METHOD PUBLIC noAction : BOOL //Return value = TRUE if busy of home and motion 
VAR_INPUT
END_VAR
home.Execute	:= FALSE;


NoAction 		:= 	NOT home.Busy ;
END_METHOD

PROPERTY PUBLIC optEnableCmdAbortedAsError : BOOL
GET
optEnableCmdAbortedAsError := Options.7;
END_GET
SET
Options.7 := optEnableCmdAbortedAsError;
END_SET
END_PROPERTY

{attribute 'monitoring' := 'call'}
PROPERTY rAdmin : REFERENCE to AxAdmin
GET
rAdmin REF= Admin;
END_GET
END_PROPERTY

{attribute 'monitoring' := 'call'}
PROPERTY rAxisRef : REFERENCE TO AXIS_REF
GET
rAxisRef REF= THIS^;
END_GET
END_PROPERTY

{attribute 'monitoring' := 'call'}
PROPERTY PUBLIC rErrHdl : REFERENCE to ERROR_HDL
GET
rErrHdl REF= ErrHdl;
END_GET
SET
ErrHdl := rErrHdl;
END_SET
END_PROPERTY

METHOD reset : Bool
VAR_INPUT
END_VAR
NoAction();
reset 			:= ErrHdl.flag OR Admin.reset(FALSE);
Event.confirm();
END_METHOD

{attribute 'monitoring' := 'call'}
PROPERTY rHome : REFERENCE To AxHoming
GET
rHome REF= Home;
END_GET
END_PROPERTY

{attribute 'monitoring' := 'call'}
PROPERTY rPara : REFERENCE TO AxPara
GET
rPara REF= Para;
END_GET
END_PROPERTY

END_FUNCTION_BLOCK

// ---- POUs/Motion/TF5100-NCI/01_Main/NCI_REF.TcPOU
{attribute 'no_check'}
FUNCTION_BLOCK NCI_REF
VAR_INPUT
	PlcToNci										AT %Q*	: PLCTONC_NCICHANNEL_REF;	//link PLC to NC
END_VAR                             				
VAR_OUTPUT                          	
	NciToPlc										AT %I*	: NCTOPLC_NCICHANNEL_REF;	//link NC to PLC

(* Extrabits out of the struct *)
	ItpRunning												:	BOOL := FALSE;	//Interpreter is running
	ItpGroupActive											:	BOOL;			//Interpreter group is active -> Axes group build 			
	GrpCnfg													:	NCI_EXT3DGROUP;	//Group configuration
	                                    					
(* ChnState *******************)        					
	IsItpChn												:	BOOL := FALSE;	//TRUE when it is interpreter channel
	IsEStopRequested										:	BOOL := FALSE;	//TRUE when EStop is requested
	IsFeedFromBackupList									:	BOOL := FALSE;	//TRUE when parameter feed comes from backup list 
	IsMovingBackward										:	BOOL := FALSE;	//TRUE when moving forward
	
(* configurated parameters of the cyclic channel *)
	PathRestWay												:	LREAL;	//remaining arc length on the current path segment
	CurrentPathSetVelo										:	LREAL;	//current path set velocity
                                        					
	SAFStatus												:	UDINT;	//SAF state
	SAFEintraege											:	UDINT;	//current number of SAF entries/tasks
	SVBStatus												:	UDINT;	//SVB state
	SVBEintraege											:	UDINT;	//current number of SVB entries/tasks
	MemLastBlockNo											:	UDINT;	//contains last block number
END_VAR
VAR
	(* NciToPlc channel extend *)
	SetCyclicLrealOffsets									:	ItpSetCyclicLRealOffsets;
	SetCyclicLrealOffsetsDone								:	BOOL;
	SetCyclicUdintOffsets									:	ItpSetCyclicUdintOffsets;
	SetCyclicUdintOffsetsDone								:	BOOL;
	
END_VAR

;

METHOD readStatus : BOOL 
VAR_INPUT
END_VAR
(* NCI Status lesen															*)
(****************************************************************************)

(****************************************************************************)
(* 4 LReal variables to configurate the interface cyclely					*)
(****************************************************************************)
	IF SetCyclicLRealOffsets.bExecute AND NOT SetCyclicLRealOffsets.bBusy
	THEN
		SetCyclicLRealOffsetsDone := NOT SetCyclicLRealOffsets.bErr;
	END_IF

	IF NOT SetCyclicLRealOffsetsDone
	THEN
		SetCyclicLRealOffsets(
			bExecute			:= NciToPlc.ChnId <> 0 AND NOT SetCyclicLRealOffsetsDone AND NOT SetCyclicLRealOffsets.bErr,
			tTimeOut			:= DEFAULT_ADS_TIMEOUT,
			nIndexOffsetParam1	:= 16#500, (* Bahnrestweg (verbleibende Bogenlaenge) auf dem aktuellen Bahnsegment *)
			nIndexOffsetParam2	:= 16#502 , (* aktuelle Bahnsollgeschwindigkeit *)
			nIndexOffsetParam3	:= ,
			nIndexOffsetParam4	:= ,
			sNciToPlc			:= NciToPlc,
			bBusy				=> ,
			bErr				=> ,
			nErrId				=> );
	END_IF

	(* reading date *)
	PathRestWay												:= NciToPlc.DoubleParams[0];	
	CurrentPathSetVelo										:= NciToPlc.DoubleParams[1];	
	//														:= NciToPlc.DoubleParams[2];	
	//														:= NciToPlc.DoubleParams[0];	

(******************************************************************************)
(* 4 DINT variables cycliaclly das Zyklsiche Interface konfigurieren						*)
(******************************************************************************)
	IF SetCyclicUdintOffsets.bExecute 
	AND NOT SetCyclicUdintOffsets.bBusy
	THEN
		SetCyclicUdintOffsetsDone 							:= NOT SetCyclicUdintOffsets.bErr;
	END_IF

	IF NOT SetCyclicUdintOffsetsDone
	THEN
		SetCyclicUdintOffsets(
			bExecute			:= NciToPlc.ChnId <> 0 AND NOT SetCyclicUdintOffsetsDone AND NOT SetCyclicUdintOffsets.bErr,
			tTimeOut			:= DEFAULT_ADS_TIMEOUT,
			nIndexOffsetParam1	:= 16#4, (* Akt SVB Status 4  *)
			nIndexOffsetParam2	:= 16#5, (* Akt SAF Status -> Running 5 *)
			nIndexOffsetParam3	:= 16#B, (* Akt Anzahl SVB Eintraege B *)
			nIndexOffsetParam4	:= 16#C, (* Akt Anzahl SAF Eintraege C *)
			sNciToPlc			:= NciToPlc,
			bBusy				=> ,
			bErr				=> ,
			nErrId				=> );
	END_IF	

	(* Daten lesen *)
	SVBStatus												:= NciToPlc.IntParams[0];	
	SAFStatus												:= NciToPlc.IntParams[1];	
	SVBEintraege											:= NciToPlc.IntParams[2];	
	SAFEintraege											:= NciToPlc.IntParams[3];	
	
(******************************************************************************)
(* Interpreterstatus lesen																		*)
(******************************************************************************)
	ItpRunning 												:= NciToPlc.ItpState > NCI_INTERPRETER_READY
																	AND NciToPlc.ItpState <> NCI_INTERPRETER_ABORTED
																	OR SAFStatus > 2
																	OR SVBStatus > 2
																	OR SAFEintraege > 0
																	OR SVBEintraege > 0;
                                							
	IF NciToPlc.BlockNo > 0 
	AND MemLastBlockNo <> NciToPlc.BlockNo
	THEN
		MemLastBlockNo 	 									:= NciToPlc.BlockNo;
	END_IF                      							
	                            							
	GrpCnfg.nXAxisId										:= NciToPlc.AcsAxisIDs[0];
	GrpCnfg.nYAxisId										:= NciToPlc.AcsAxisIDs[1];
	GrpCnfg.nZAxisId										:= NciToPlc.AcsAxisIDs[2];
	GrpCnfg.nQ1AxisId										:= NciToPlc.AcsAxisIDs[3];
	GrpCnfg.nQ2AxisId										:= NciToPlc.AcsAxisIDs[4];
	GrpCnfg.nQ3AxisId										:=	NciToPlc.AcsAxisIDs[5];
	GrpCnfg.nQ4AxisId										:= NciToPlc.AcsAxisIDs[6];
	GrpCnfg.nQ5AxisId										:= NciToPlc.AcsAxisIDs[7];
                                							
	ItpGroupActive											:= GrpCnfg.nXAxisId <> 0
																	OR GrpCnfg.nYAxisId <> 0
																	OR GrpCnfg.nZAxisId <> 0
																	OR GrpCnfg.nQ1AxisId <> 0
																	OR GrpCnfg.nQ2AxisId <> 0
																	OR GrpCnfg.nQ3AxisId <> 0
																	OR GrpCnfg.nQ4AxisId <> 0
																	OR GrpCnfg.nQ5AxisId <> 0;
                                	
(******************************************************************************)
(* Channelstatus lesen																			*)
(******************************************************************************)
	IsItpChn												:= NciToPlc.ChnState.0;
	IsEStopRequested										:= NciToPlc.ChnState.8;
	IsFeedFromBackupList									:= NciToPlc.ChnState.10;
	IsMovingBackward										:= NciToPlc.ChnState.11;

	
(* ENUM ItpMode
	0x0	Defaultbelegung (Abwahl der übrigen Betriebsarten)
	0x1	Einzelsatzbetrieb im NC-Kern (Satzausführungstask/SAF)
	0x1000	reserviert
	0x2000	reserviert
	0x4000	Einzelsatzbetrieb im Interpreter
*)

(* ItpStatus
ITP_STATE_IDLE  The interpreter is in idle state when there is no NC program loaded as yet or when a group reset is being executed.
The interpreter also goes into idle state when a current program is stopped. In the case a group reset must be executed in order to prevent error 0x42C5. 
It is therefore recommended to execute a group reset after stopping via the PLC.
 
ITP_STATE_READY  After successful loading of an NC program, the interpreter is in ready state.
After a program has been successfully processed and exited, the interpreter goes into ready state. 
In the meantime, however, other states are accepted.  
 
ITP_STATE_ABORTED  Tritt während der Abarbeitung des NC Programms ein Laufzeitfehler auf, 
so geht der Interpreter in den Aborted eSTATE. Der eigentliche Fehlercode ist dem Kanal Status zu entnehmen.  

ITP_STATE_SINGLESTOP  If a run time error occurs during the processing of an NC program, the interpreter goes into aborted state. The actual error code is given in Channel Status.
 
NCI_INTERPRETER_INITFAILED:	UDINT	:=	0;
NCI_INTERPRETER_IDLE:			UDINT	:=	1;
NCI_INTERPRETER_READY:			UDINT	:=	2;
NCI_INTERPRETER_STARTED:		UDINT	:=	3;
NCI_INTERPRETER_SCANNING:		UDINT	:=	4;
NCI_INTERPRETER_RUNNING:		UDINT	:=	5;
NCI_INTERPRETER_STAY_RUNNING:	UDINT	:=	6;
NCI_INTERPRETER_WRITETABLE:		UDINT	:=	7;
NCI_INTERPRETER_SEARCHLINE:		UDINT	:=	8;
NCI_INTERPRETER_END:			UDINT	:=	9;
NCI_INTERPRETER_SINGLESTOP:		UDINT	:=	10;
NCI_INTERPRETER_ABORTING:		UDINT	:=	11;
NCI_INTERPRETER_ABORTED:		UDINT	:=	12;
NCI_INTERPRETER_FAULT:			UDINT	:=	13;
NCI_INTERPRETER_RESET:			UDINT	:=	14;
NCI_INTERPRETER_STOP:			UDINT := 15;
NCI_INTERPRETER_WAITFUNC:		UDINT	:=	16;
NCI_INTERPRETER_FLUSHBUFFERS:	UDINT	:=	17;

*)

	readStatus											:= TRUE;
(******************************************************************)
END_METHOD

END_FUNCTION_BLOCK

// ---- POUs/Motion/TF511x-KIN/01_Main/KinAdmin.TcPOU
//Kinematic group administration - Enable/Disable/Reset group
//based on TF511x - Tc2_NcKinematicTransformation
//ACS - Axis coordinate system => Robot motors M1-Mx 
//MCS - Machine coordinate system >= Cartesian Axis X,Y,Z,Rx,Ry,Rz (A,B,C) 
FUNCTION_BLOCK KinAdmin
VAR_INPUT
	ResetTrig												:	BOOL := FALSE;
	Enable													:	BOOL := FALSE; (* TRUE = Build Group , FALSE = Reconfig Group *)
	Override												:	LREAL	:= 0.0;
	ItpChannelId 											: 	UDINT := 0; (* Bei 0 wirtd der ITP Kanal nicht resetet *)
	AxesList												: 	ST_KinAxes;
	rKINRef													:	REFERENCE TO KIN_REF := 0;
END_VAR
VAR_IN_OUT
END_VAR
VAR_OUTPUT
	Busy													:	BOOL;
	Done													:	BOOL;
	Error													:	BOOL;
{attribute 'displaymode':='hex'}
	ErrorId													:	UDINT;
	ErrorText												:	STRING(40);
END_VAR
VAR
(* cache **************************************************************************)
	MemDone													:	BOOL;
	MemFnc													:	INT := 1;
	                        								
(* MC-functonblock instances *******************************************************)
	ResetKinGroup											: 	FB_KinResetGroup ;
	ConfigKinGroup											:	FB_KinConfigGroup  ;

(* Dummy Speicher **********************************************************)
	OK 														: BOOL;
END_VAR

	(* Kinematic group administration										*)
	(************************************************************************)

(* aborting function-block call if pointer is not valid ****************************************)
IF NOT __ISVALIDREF(rKINRef) 
THEN
	Busy													:= NOT Error;
	ErrorId													:= E_AdsErr.DEVICE_INVALIDPARM;
	Error													:= TRUE;
	Done													:= FALSE;
	ErrorText												:= 'Reference to rKINRef invalid (0)';
	RETURN;
END_IF

(* reading axis-status from NCtoPLC-channel ***************************************************)
	rKINRef.readStatus();

(* accepting setvalue-barrier e.g. for hardware limit switch **********************************)
	rKINRef.PlcToNci.ChnAxesOvr 							:= LREAL_TO_DWORD(LIMIT(0.0,Override,100.0) * 10000.0 );

(* ctrl programm ******************************************************************************)
	ConfigKinGroup.bExecute									:=	NOT ConfigKinGroup.bBusy
																AND(
																Enable
																AND NOT ConfigKinGroup.bCartesianMode
																OR
																NOT Enable
																AND ConfigKinGroup.bCartesianMode);

	IF ConfigKinGroup.bExecute
	THEN
		ConfigKinGroup.bCartesianMode						:= Enable;
	END_IF

	ConfigKinGroup(
		bExecute		:= ,
		bCartesianMode	:= ,
		stAxesList		:= AxesList,
		stKinRefIn		:= rKinRef.NciToPlc,
		bBusy			=> ,
		bDone			=> ,
		bError			=> ,
		nErrorId		=> );

(* Reset Grp ****************************************************************)
	IF Memfnc < 0
	THEN
		IF ResetTrig
		THEN
			reset(Execute:= TRUE);
			MemFnc											:= 1;
		END_IF
	ELSIF NOT reset(Execute:= ResetTrig)
	THEN
		MemFnc												:= -1;
	END_IF

(******************************************************************************)
(* Ctrl Status 																					*)
(******************************************************************************)
	Busy						:= ResetKinGroup.bBusy OR ConfigKinGroup.bBusy;
	
	IF Busy
	THEN
		Error												:= FALSE;
		ErrorId												:= 0;
		ErrorText											:= '';
	ELSIF ConfigKinGroup.bError
	THEN
		Error												:= TRUE;
		ErrorId												:= ConfigKinGroup.nErrorID;
		ErrorText											:= CONCAT('ConfigKinGroup ErrorId: ', UDINT_TO_STRING(Errorid));
	ELSIF ResetKinGroup.bExecute
		AND ResetKinGroup.bError
	THEN
		Error												:= TRUE;
		ErrorId												:= ResetKinGroup.nErrorID;
		ErrorText											:= CONCAT('ResetKinGroup ErrorId: ', UDINT_TO_STRING(Errorid));
	ELSIF rKINRef.NciToPlc.ErrorCode <> 0
	THEN
		Error												:= TRUE;
		ErrorId												:= rKINRef.NciToPlc.ErrorCode;
		ErrorText											:= CONCAT('KIN Grp ErrorId: ', UDINT_TO_STRING(Errorid));
	ELSE
		Error												:= FALSE;
		ErrorId												:= 0;
		ErrorText											:= '';
	END_IF

	IF ResetKinGroup.bDone
		OR ConfigKinGroup.bDone
	THEN
		MemDone												:= TRUE;
	END_IF

	Done													:= NOT Busy AND MemDone;

	IF done
	THEN
		MemDone												:= FALSE;
	END_IF

(**************************************************************************************************)

METHOD PUBLIC reset : BOOL //Return value = TRUE if busy
//required parameter
//rKinRef
//ItpChannelId
//AxesList
VAR_INPUT
	Execute													:	BOOL;
END_VAR
IF NOT __ISVALIDREF(rKINRef) THEN
	Busy													:= NOT Error;
	ErrorId													:=E_AdsErr.DEVICE_INVALIDPARM;
	Error													:= TRUE;
	Done													:= FALSE;
	ErrorText												:= 'Reference to rKINRef  invalid (0)';
	RETURN;
END_IF

	IF Execute
	THEN
		Error												:=	FALSE;
		ErrorId												:= 0;
		ResetKinGroup.bExecute 								:= rKinRef.NciToPlc.ErrorCode <> 0;
	ELSIF NOT ResetKinGroup.bBusy
	THEN
		Error												:=	FALSE;
		ErrorId												:= 0;
		ResetKinGroup.bExecute 								:= FALSE;

	END_IF

	ResetKinGroup(
		bExecute		:= ,
		nItpChannelId	:= ItpChannelId,
		stKinRefIn		:= rKinRef.NciToPlc,
		stAxesList		:= AxesList,
		bBusy			=> Busy,
		bDone			=> ,
		bError			=> ,
		nErrorId		=> );

	Done													:= NOT ResetKinGroup.bBusy
																AND NOT ResetKinGroup.bError
																AND ResetKinGroup.bExecute;

	IF NOT Busy
	THEN
		IF ResetKinGroup.bExecute
		THEN
			Error											:=	ResetKinGroup.bError;
			ErrorId											:= ResetKinGroup.nErrorId;
			ErrorText										:= SEL(Error , '' ,  CONCAT('Error ResetKinGroup id: ',  UDINT_TO_STRING(Errorid)));
		END_IF
		IF NOT Execute
		THEN
			MemFnc											:= -1 ;
			ResetKinGroup(	bExecute := FALSE, 
							stKinRefIn := rKinRef.NciToPlc, 
							stAxesList := AxesList);
		END_IF
	END_IF
	
	reset													:= Busy;
END_METHOD

END_FUNCTION_BLOCK

// ---- POUs/Motion/TF511x-KIN/01_Main/KIN_REF.TcPOU
//Kinematic group ref - call ReadStatus cyclic
FUNCTION_BLOCK KIN_REF
VAR_INPUT
	PlcToNci										AT %Q*	:	PLCTONC_NCICHANNEL_REF;
END_VAR                     						
VAR_OUTPUT                  						
	NciToPlc										AT %I*	:	NCTOPLC_NCICHANNEL_REF;
                            						
	ChnOperationState										:	E_KINSTATUS := 0;
	CartesianModeON											:	BOOL := FALSE;
	                                					
(* ChnState ***************************)
	IsKinematicChn											:	BOOL := FALSE;
	                                					
	AxList													: ST_KinAxes;
END_VAR
VAR
END_VAR

;

METHOD PUBLIC readStatus : booL;
VAR_INPUT
END_VAR
(* Kin Channel State *********************************************************)
	F_KinGetAcsMcsAxisIds(AxList,NciToPlc);
	
	ChnOperationState 										:= TO_INT(F_KinGetChnOperationState(NciToPlc));

	CartesianModeON											:= NciToPlc.AcsAxisIDs[0] <> 0 AND NciToPlc.AcsAxisIDs[1] <> 0;
	
	IsKinematicChn											:= NciToPlc.ChnState.1;

	readStatus												:= TRUE;
(*****************************************************************************)
END_METHOD

END_FUNCTION_BLOCK

// ---- POUs/Motion/TF511x-KIN/02_Options/KinLockUnlockTrafoParam.TcPOU
//Lock or Unlock kinematic group parameter
FUNCTION_BLOCK KinLockUnlockTrafoParam
VAR_INPUT
	Execute													:	BOOL	:= FALSE;
	Lock													:	BOOL 	:= TRUE;
   	oidTrafo												:	UDINT;
END_VAR                     								
VAR_OUTPUT                  								
	Busy													:	BOOL	:= FALSE;
	Done													:	BOOL	:= FALSE;
	Error													:	BOOL	:= FALSE;
	ErrorId													:	UDINT	:= 0;
END_VAR                     								
VAR                         	
	State													:	UDINT	:= 0;
	ADSWRITE												:	ADSWRITE;
END_VAR

CASE State OF
0:
	Done													:= FALSE;
	Error													:= FALSE;
	ErrorId													:= 0;
	Busy 													:= FALSE;
	
	IF Execute THEN
		AdsWrite(WRITE := FALSE);
		AdsWrite(
			NETID		:='',
			PORT		:= 10,
			IDXGRP		:=oidTrafo,
			IDXOFFS		:=SEL(Lock, 16#05030210, 16#0503020F),
			LEN			:= 0,
			SRCADDR		:=0 ,
			WRITE		:= TRUE,
			TMOUT		:= DEFAULT_ADS_TIMEOUT,
			BUSY		=> ,
			ERR			=> ,
			ERRID		=> );

		Busy												:= TRUE;
		State												:= 10;
	END_IF
10:
	AdsWrite(
		TMOUT	:= DEFAULT_ADS_TIMEOUT,
		BUSY	=>,
		ERR		=>Error,
		ERRID	=>ErrorId);
		
	IF NOT AdsWrite.BUSY 
	THEN
		IF NOT AdsWrite.ERR 
		THEN
			Done											:= TRUE;
		END_IF
		IF NOT Execute THEN
			State											:= 0;
		ELSE
			State											:= 20;
		END_IF
		AdsWrite(WRITE:=FALSE);
	END_IF
20:
	Busy													:= FALSE;
	IF NOT Execute THEN
		State												:= 0;
	END_IF

END_CASE

END_FUNCTION_BLOCK

// ---- POUs/Motion/TF50xx-NC/02_Options/Coupling/AxFlyingSaw.TcPOU
{attribute 'no_check'}
//Nc-axis flying saw control
//based on Tc2_MC2_FlyingSaw library
FUNCTION_BLOCK AxFlyingSaw EXTENDS AxFbBase
VAR_OUTPUT CONSTANT
	FNC_GEAR_OUT											:	INT := 0;
	FNC_GEAR_IN_VELO										:	INT := 1;
	FNC_GEAR_IN_POS											:	INT := 2;
END_VAR                     								
VAR_INPUT                   								
	Fnc														:	INT (FNC_GEAR_OUT..FNC_GEAR_IN_POS) := FNC_GEAR_OUT;
	RatioNumerator											:	LREAL := 1.0; (* Getriebefaktor Numerator/Zähler *)
	RatioDenominator										:	UINT := 1; (* Getriebefaktor Denominator/Nenner *)
	MasterSyncPosition										: 	LREAL := 0.0;
	SlaveSyncPosition										: 	LREAL := 0.0;
	MasterStartDistance										: 	LREAL := 0.0;
	SyncMode												: 	ST_SyncMode; (*... mode ...
																						GearInSyncMode : E_GearInSyncMode;
                            								
																					... 32 bit check mask ... 
																						GearInSync_CheckMask_MinPos : BOOL;
																						GearInSync_CheckMask_MaxPos : BOOL;
																						GearInSync_CheckMask_MaxVelo : BOOL;
																						GearInSync_CheckMask_MaxAcc : BOOL;
																						GearInSync_CheckMask_MaxDec : BOOL;
																						GearInSync_CheckMask_MaxJerk : BOOL;
																						GearInSync_CheckMask_OvershootPos : BOOL;
																						GearInSync_CheckMask_UndershootPos : BOOL;
																						GearInSync_CheckMask_OvershootVelo : BOOL;
																						GearInSync_CheckMask_UndershootVelo : BOOL;
																						GearInSync_CheckMask_OvershootVeloZero : BOOL;
																						GearInSync_CheckMask_UndershootVeloZero : BOOL;
																				
																					... operation masks ...
																						GearInSync_OpMask_RollbackLock : BOOL;
																						GearInSync_OpMask_InstantStopOnRollback : BOOL;
																						GearInSync_OpMask_PreferConstVelo : BOOL;
																						GearInSync_OpMask_IgnoreMasterAcc : BOOL;*)
	Velo													:	LREAL := 0.0;	(* Flying Saw ... Max Slave-Geschwindigkeit in Synchronisierungsphase. Bei 0 --> Systemmanager-Daten. Achtung: Geschwindigkeit wird nur überprüft, wenn die Überprüfung mit der Variablen SyncMode aktiviert wird.*)
	Acc														:	LREAL := 0.0; (* Bei 0 werden wird die Beschleunigung aus dem TCManager uebernommen *)
	Dec														:	LREAL := 0.0; (* Bei 0 werden wird die Verzoegerung aus dem TCManager uebernommen *)
	Jerk													:	LREAL := 0.0; (* Bei 0 werden wird der Ruck aus dem TCManager uebernommen *)
(*	BufferMode												:	MC_BufferMode := MC_Aborting;(* 	MC_Aborting,
																												MC_Buffered,
																												MC_BlendingLow,
																												MC_BlendingPrevious,
																												MC_BlendingNext,
																												MC_BlendingHigh *)
*)                          								
(*	Options 												: 	ST_MOVEOptions; *)
//	rCamTableCharac 										:  REFERENCE TO MC_FlyingSawCharacValues; (* Struktur mit den charakteristischen Kennwerten.*)
	rMasterAxis												:	REFERENCE TO AXIS_REF := 0;
END_VAR                     								
VAR_IN_OUT                  								
END_VAR                     								
VAR_OUTPUT                  								
	StartSync 												:  BOOL;  (* Flying Saw*)
END_VAR
VAR
(* cache **************************************************************************)
	MemFnc													:	INT := -1;
                            								
(* timer *)                 								
                            	
(* trigger *)               	
                            	
(* MC-function-block instances *****************************************************)
	MC_GearOut												:	MC_GearOut;
	MC_GearInVelo 											:  MC_GearInVelo;
	MC_GearInPos											:  MC_GearInPos;	
//	MC_ReadCharacteristics									:  MC_ReadFlyingSawCharacteristics; (* charakteristischen Kennwerte der Synchronisierungsphase ausgelesen *)

(* Dummy storage *******************************************************************)
(*	i,j		: INT := 0 ; *)
	Dummy 	: BOOL; 
END_VAR

	(************************************************************************************)
	(*																					*)
	(*		B E C K H O F F   N E W   A U T O M A T I O N   T E C H N O L O G Y    		*)
	(*																					*)
	(*		Eiserstr.5	D-33415 Verl	Germany	phone:	+49-5246-0	www.Beckhoff.Com	*)
    (*																					*)
    (*		Bausteinbeschreibung	:	Flying Saw Achs Baustein						*)
	(*		TwinCAT-Version			:	3.x or higher									*)
	(*		Version					:	V3.0 / 03/13									*)
	(*		Lib						:	TcMC2_FlyingSaw.lib 							*)
 	(*		Autor					:	DS												*)
	(*																					*)
	(************************************************************************************)

(* Execute ***************************************************************************************)
	rtExecute(CLK := Execute);
	IF rtExecute.Q
		AND MemFnc < 0
	THEN
		MemFnc 												:= Fnc ;
		Busy												:= TRUE;
		Done												:= FALSE;
		Error												:= FALSE;
		ErrorID												:= 0;
		CmdAborted											:= FALSE;
		ErrorText											:= '';
	END_IF

(* Call Method ***********************************************************************************)
	CASE MemFnc OF
	FNC_GEAR_OUT:
		GearOut(Execute);

	FNC_GEAR_IN_VELO:
		GearInVelo(Execute);

	FNC_GEAR_IN_POS:
		GearInPos(Execute);

	-1:
		IF NOT Execute
		THEN
			StartSync										:= FALSE;
			Busy											:= FALSE;
			Done											:= FALSE;
			Error											:= FALSE;
			ErrorID											:= 0;
			CmdAborted										:= FALSE;
			ErrorText										:= '';
		END_IF                          					
	ELSE                                					
		StartSync											:= FALSE;
		Busy												:= FALSE;
		Done												:= FALSE;
		Error												:= Execute;
		ErrorID												:= E_AdsErr.DEVICE_INVALIDPARM;
		CmdAborted											:= FALSE;
		ErrorText											:= CONCAT('invalid parameter value(s) Fnc no: ' , INT_TO_STRING(MemFnc));
	END_CASE

(*************************************************************************************************)

METHOD PUBLIC gearInPos : BOOL //Return value = TRUE if busy
//required parameter
//rAxis
//rMasterAxis
//RatioNumerator
//RatioDenominator
//MasterSyncPosition
//SlaveSyncPosition
//SyncMode
//MasterStartDistance
//Velo
//Acc
//Dec
//Jerk
VAR_INPUT
	Execute													:	BOOL;
END_VAR
MemFnc														:= FNC_GEAR_IN_POS;
THIS^.Execute												:= Execute;
	
IF NOT __ISVALIDREF(rAxis) 
THEN
	Busy													:= NOT Error;
	Error													:= TRUE;
	ErrorId													:= E_AdsErr.DEVICE_INVALIDPARM;
	CmdAborted												:= FALSE;
	Done													:= FALSE;
	Active													:= FALSE;
	ErrorText												:= 'Reference rAxis invalid (0)';
	MemFnc													:= SEL(Execute , -1 ,MemFnc); 
	RETURN;
ELSIF NOT __ISVALIDREF(rMasterAxis)
THEN
	Busy													:= NOT Error;
	Error													:= TRUE;
	ErrorId													:= E_AdsErr.DEVICE_INVALIDPARM;
	CmdAborted												:= FALSE;
	Done													:= FALSE;
	ErrorText												:= 'Reference rMasterAxis invalid (0)';
	MemFnc													:= SEL(Execute , -1 ,MemFnc); 
	RETURN;
END_IF

	MC_GearInPos(
		Execute				:= Execute,
		RatioNumerator		:= RatioNumerator,
		RatioDenominator	:= RatioDenominator,
		MasterSyncPosition	:= MasterSyncPosition,
		SlaveSyncPosition	:= SlaveSyncPosition,
		SyncMode			:= SyncMode,
		MasterStartDistance	:= MasterStartDistance,
		Velocity			:= Velo,
		Acceleration		:= Acc,
		Deceleration		:= Dec,
		Jerk				:= Jerk,
		BufferMode			:= ,
		Options				:= ,
		Master				:= rMasterAxis,
		Slave				:= rAxis,
		StartSync			=> StartSync,
		InSync				=> Done,
		Busy				=> Busy,
		Active				=> Active,
		CommandAborted		=> CmdAborted,
		Error				=> Error,
		ErrorID				=> ErrorID);
		
	

	IF Error THEN
		LastErrorId											:= ErrorId;
		ErrorText 											:= CONCAT('MC_GearInPos ID:' , UDINT_TO_STRING(ErrorId));
	ELSE
		ErrorText 											:= '';
	END_IF

	IF NOT Execute AND NOT Busy
	THEN
		MemFnc												:= -1;
	END_IF
	
	GearInPos												:= Busy;
END_METHOD

METHOD PUBLIC gearInVelo : BOOL //Return value = TRUE if busy
//required parameter
//rAxis
//rMasterAxis
//RatioNumerator
//RatioDenominator
//SyncMode
//Velo
//Acc
//Dec
//Jerk
VAR_INPUT
	Execute													:	BOOL;
END_VAR
MemFnc														:= FNC_GEAR_IN_VELO;
THIS^.Execute												:= Execute;
	
IF NOT __ISVALIDREF(rAxis)
THEN
	Busy													:= NOT Error;
	Error													:= TRUE;
	ErrorId													:= E_AdsErr.DEVICE_INVALIDPARM;
	CmdAborted												:= FALSE;
	Done													:= FALSE;
	Active													:= FALSE;
	ErrorText												:= 'Reference rAxis invalid (0)';
	MemFnc													:= SEL(Execute , -1 ,MemFnc); 
	RETURN;
ELSIF NOT __ISVALIDREF(rMasterAxis)
THEN
	Busy													:= NOT Error;
	Error													:= TRUE;
	ErrorId													:= E_AdsErr.DEVICE_INVALIDPARM;
	CmdAborted												:= FALSE;
	Done													:= FALSE;
	ErrorText												:= 'Reference rMasterAxis invalid (0)';
	MemFnc													:= SEL(Execute , -1 ,MemFnc); 
	RETURN;
END_IF

	MC_GearInVelo(
		Execute			:= Execute,
		RatioNumerator	:= RatioNumerator ,
		RatioDenominator:= RatioDenominator ,
		SyncMode		:= SyncMode,
		Velocity		:= Velo,
		Acceleration	:= Acc,
		Deceleration	:= Dec,
		Jerk			:= Jerk,
		BufferMode		:= ,
		Options			:= ,
		Master			:= rMasterAxis,
		Slave			:= rAxis,
		StartSync		=> StartSync,
		InSync			=> Done,
		Busy			=> Busy,
		Active			=> Active,
		CommandAborted	=> CmdAborted,
		Error			=> Error,
		ErrorID			=> ErrorId);
	
	IF Error THEN
		LastErrorId											:= ErrorId;
		ErrorText 											:= CONCAT('MC_GearInVelo ID:' , UDINT_TO_STRING(ErrorId));
	ELSE
		ErrorText 											:= '';
	END_IF

	IF NOT Execute AND NOT Busy
	THEN
		MemFnc												:= -1;
	END_IF
	
	GearInVelo												:= Busy;
END_METHOD

METHOD PUBLIC gearOut : BOOL //Return value = TRUE if busy
//required parameter
//rAxis
VAR_INPUT
	Execute													:	BOOL;
END_VAR
MemFnc														:= FNC_GEAR_OUT;
THIS^.Execute												:= Execute;

IF NOT __ISVALIDREF(rAxis) 
THEN
	Busy													:= NOT Error;
	Error													:= TRUE;
	ErrorId													:= E_AdsErr.DEVICE_INVALIDPARM;
	CmdAborted												:= FALSE;
	Done													:= FALSE;
	Active													:= FALSE;
	ErrorText												:= 'Reference rAxis invalid (0)';
	MemFnc													:= SEL(Execute , -1 ,MemFnc); 
	RETURN;
END_IF

	MC_GearOut(
		Execute	:= Execute,
		Options	:= ,
		Slave	:= rAxis,
		Done	=> Done,
		Busy	=> Busy,
		Error	=> Error,
		ErrorID	=> ErrorID);

	Active													:= Busy;
	CmdAborted												:= FALSE;
	StartSync												:= FALSE;
	
	IF Error THEN
		LastErrorId											:= ErrorId;
		ErrorText 											:= CONCAT('MC_GearOut ID:' , UDINT_TO_STRING(ErrorId));
	ELSE
		ErrorText 											:= '';
	END_IF

	IF NOT Execute AND NOT Busy
	THEN
		MemFnc												:= -1;
	END_IF                  								
                            	
	GearOut													:= Busy;
END_METHOD

END_FUNCTION_BLOCK

// ---- POUs/Motion/TF50xx-NC/02_Options/Error/AxNcEventHandling.TcPOU
{attribute 'no_check'}
FUNCTION_BLOCK AxNcEventHandling
VAR CONSTANT
END_VAR     
VAR_INPUT
	Flag													:	BOOL := FALSE;  
	ConfirmTrig													:	BOOL := FALSE;
	MsgId													:	UDINT := 201; //Default
	SourceId												:	UDINT := 101000; //TwinCat-NC axis default multisource Id + Ax id for detailed event message
	AxisId													:	UDINT := 0;
	ErrorID													:	UDINT := 0; (* NC Error Id Bsp 18000 -Drive Error *)
	Name													: 	STRING(30) := '';
END_VAR                         							
VAR_OUTPUT                      							
	State													:	UDINT := TCEVENTSTATE_INVALID;
																		(* TCEVENTSTATE_INVALID  	: WORD := 16#0000; (* Ungültig, kommt auch wenn Event noch nicht gemeldet. *)
																			TCEVENTSTATE_SIGNALED  	: WORD := 16#0001; (* Event ist gemeldet, aber weder gegangen noch quittiert. *)
																			TCEVENTSTATE_RESET  		: WORD := 16#0002; (* Event ist abgemeldet ('gegangen'). *)
																			TCEVENTSTATE_CONFIRMED  : WORD := 16#0010 (16); (* Event ist quittiert. *)
																			TCEVENTSTATE_RESETCON  	: WORD := 16#0012 (17); (* Event ist abgemeldet und quittiert *) *)
{attribute 'displaymode':='binary'}
	Status													:	DWORD; (*	.0 - .8 = event <class id>  / .15 Quit required / .16 = Level 0 , .17 = Level 1 , .18 = Level 2, .......... / .31 active
																			TCEVENTCLASS_NONE			:=0,	(* No class *)
																			TCEVENTCLASS_MAINTENANCE	:=1,	(* Maintenance hint *)
																			TCEVENTCLASS_MESSAGE		:=2,	(* Message *)
																			TCEVENTCLASS_HINT			:=3,	(* Hint *)
																			TCEVENTCLASS_STATEINFO		:=4,	(* State information *)
																			TCEVENTCLASS_INSTRUCTION	:=5,	(* Instruction *)
																			TCEVENTCLASS_WARNING		:=6,	(* Warning *)
																			TCEVENTCLASS_ALARM			:=7,	(* Alarm *)
																			TCEVENTCLASS_PARAMERROR		:=8		(* Parameter error *)  *)
END_VAR
VAR
	AdsEvent												:		ADSLOGEVENT :=(
																		Event			:= FALSE,
																		NETID			:= '',
																		PORT			:= AMSPORT_EVENTLOG,
																		TMOUT 			:= DEFAULT_ADS_TIMEOUT,
																		EventConfigData := (
																					Class 			:= TC2_SYSTEM.TCEVENTCLASS_ALARM,
																					Prio 			:= TCEVENTPRIO_IMPLICIT,
																					ProgId 			:= 'TcEventFormatter.TcXmlFormatter',
																					Flags 			:= 16#0140 (* TCEVENTFLAG_LOG OR TCEVENTFLAG_SRCID *),
																					StreamType 		:= TCEVENTSTREAM_NORMAL (* TCEVENTSTREAM_SIMPLE *),
																					bQuitRequired 	:= FALSE));
                    										
	FormatString 											: STRING(15) := '%s%d%s%s%d%s';
                    										
	pParaArray												: ARRAY [1..6] OF PVOID;
                    										
	Para1													: STRING(30);
	Para2													: UDINT;
	Para3													: STRING(70);
	Para4													: STRING(70);
	Para5													: UDINT;
	Para6													: STRING(20);
	SetClass												: E_TcEventClass := TC2_SYSTEM.TCEVENTCLASS_ALARM;
END_VAR

(* Send axis error text to EventLogger		 							*)
(************************************************************************)

(* Event Config ************************************************)
	IF Status.31 //Message active
	THEN (* work EventLogger *)

		AdsEvent(
			NETID			:= ,(* siehe deklaration *)
			PORT			:= ,(* siehe deklaration *)
			Event			:= NOT AdsEvent.FbCleanup AND(Flag AND Para2 = ErrorID OR AdsEvent.EventState = TCEVENTSTATE_INVALID AND NOT AdsEvent.Quit),
			EventQuit		:= AdsEvent.EventState <> TCEVENTSTATE_INVALID
								AND AdsEvent.EventConfigData.bQuitRequired
								AND NOT AdsEvent.Eventstate.4
								AND NOT AdsEvent.Quit
								AND(
								ConfirmTrig
								OR Para2 <> ErrorID
								OR AdsEvent.EventQuit), (* quit send *)
			EventConfigData	:= ,(* siehe deklaration *)
			EventDataAddress:= ADR(pParaArray),
			EventDataLength	:= ,
			FbCleanup		:= NOT AdsEvent.FbCleanup AND(AdsEvent.Err OR AdsEvent.EventState = TCEVENTSTATE_RESETCON),
			TMOUT			:= ,(* siehe deklaration *)
			EventState		=> ,
			Err				=> ,
			ErrId			=> ,
			Quit			=> );

		IF AdsEvent.Event
			AND AdsEvent.EventState = TCEVENTSTATE_INVALID
		THEN
			State 											:= SEL(Flag, TCEVENTSTATE_RESET, TCEVENTSTATE_SIGNALED);
		ELSIF AdsEvent.Quit
			AND AdsEvent.EventState = TCEVENTSTATE_INVALID
			AND AdsEvent.EventQuit
			OR 
			AdsEvent.FbCleanup		
		THEN
			State 											:= TCEVENTSTATE_RESETCON;
		ELSIF(AdsEvent.Err OR NOT AdsEvent.Event AND AdsEvent.EventState = TCEVENTSTATE_INVALID)
			AND_THEN Gvl.EventHandlingStatistic.CountOut(Status)
		THEN
			State											:= TCEVENTSTATE_INVALID;
		ELSE
			State											:= MAX(State, AdsEvent.EventState);
		END_IF
	
	ELSIF flag AND SourceId > 0
	THEN (* fire event *)
	(*	Type : 2 - Axis Event 201
		%1 User Name 
		%2 	Unique error id (DINT)
		%3	Error text (STRING) ) Bsp.: [S750E20392]
		@V1:%4	Error description (STRING) Bsp.: [S751E20392]
		%5	Logical axis id (DINT)
		@V2:%6	Position OF axis (REAL) or Reserved text 
	
	*)
		Para1 												:= Name;
		Para2 												:= ErrorID;
              												
		Para3 												:= CONCAT('[S','700'); (* SOURCE_TEXT_PTPNCI = 701 *)
		Para3 												:= CONCAT(Para3,'E');
		Para3 												:= CONCAT(Para3,UDINT_TO_STRING(ErrorID));
		Para3 												:= CONCAT(Para3,']');
              												
		Para4 												:= CONCAT('[S','701'); (* SOURCE_DESC_PTPNCI = 701 *)
		Para4 												:= CONCAT(Para4,'E');
		Para4 												:= CONCAT(Para4,UDINT_TO_STRING(ErrorID));
		Para4 												:= CONCAT(Para4,']');
              												
		Para5 												:= AxisId;
		Para6 												:= ''; (* Reserve *)

		pParaArray[1] 										:= ADR(Para1);
		pParaArray[2] 										:= ADR(Para2);
		pParaArray[3] 										:= ADR(Para3);
		pParaArray[4] 										:= ADR(Para4);
		pParaArray[5] 										:= ADR(Para5);
		pParaArray[6] 										:= ADR(Para6);

		
		AdsEvent.EventConfigData.Id 						:= MsgId; (* MSG_ID = 201 *)
 		AdsEvent.EventConfigData.DataFormatStrAddress 		:= ADR(FormatString);
		AdsEvent.EventConfigData.SourceId 					:= SourceId + AxisId;
		Status												:= Gvl.EventHandlingStatistic.InitEvent(SetClass , AdsEvent.EventConfigData);	

		IF AdsEvent.Err AND NOT AdsEvent.FbCleanup
		THEN
			AdsEvent(
				Event			:= FALSE,
				EventQuit 		:= FALSE,
				EventDataAddress:= ADR(pParaArray),
				FbCleanup		:= TRUE,
				EventState		=> );
		
		ELSE (* Fire Event *)
			AdsEvent( 	Event			:= FALSE,
						EventQuit 		:= FALSE, 
						FbCleanup 		:= FALSE, 
						EventDataAddress:= ADR(pParaArray));
			AdsEvent( 	Event 	:= TRUE);			
			IF NOT AdsEvent.Err AND_THEN Gvl.EventHandlingStatistic.CountIn(Status) //Add event to statistic and continue if added successfully
			THEN			
				State 										:= TCEVENTSTATE_SIGNALED;
			END_IF
		END_IF
	END_IF

(*****************************************************************)

END_FUNCTION_BLOCK

// ---- POUs/Motion/TF50xx-NC/03_Utilities/getOvrVelo.TcPOU
{attribute 'no_check'}
//Override function - Returns velocity setpoint based on max velo and requested override 
FUNCTION getOvrVelo : LREAL
VAR_INPUT
	SetVelo													:	LREAL;
	MaxVelo													:	LREAL;
END_VAR
VAR
END_VAR

IF 	MaxVelo = 0.0 OR SetVelo = 0.0
THEN
	GetOvrVelo 												:= 0.0;
ELSE                										
	GetOvrVelo 												:= 100.0 / MaxVelo * SetVelo;
END_IF

END_FUNCTION

// ---- POUs/StringHelper/getCntCharInWStr.TcPOU
{attribute 'no_check'}
//Returns the count of a particular char found in a string line
FUNCTION getCntCharInWStr : INT
VAR_INPUT
	Char													:	WSTRING(3):=";";
	Strline													:	WSTRING(MAX_STRING_LENGTH);
END_VAR             										
VAR                 
	tmpString												:	WSTRING(MAX_STRING_LENGTH) ;										
	pos,k													:	INT;
END_VAR

IF Strline <> "" AND Char <> ""
THEN	
	MEMSET(ADR(tmpString),0,SIZEOF(tmpString));
	MEMCPY(ADR(tmpString),ADR(Strline),TO_UDINT(WLEN(Strline) * 2));
	pos 													:= WFIND (tmpString,char);
	WHILE pos <> 0 DO		
		k													:=  pos + (WLEN(char) - 1);
		tmpString											:=	WRIGHT(tmpString,WLEN(tmpString) - k);
		pos 												:= 	WFIND (tmpString,char);
		getCntCharInWStr									:=	getCntCharInWStr+1;
	END_WHILE;
ELSE
	getCntCharInWStr										:= 0;
END_IF

END_FUNCTION

// ---- POUs/StringHelper/HEXSTR_TO_DWORD.TcPOU
{attribute 'no_check'}
//Converts a hex string into a 32 bit DWORD number
FUNCTION HEXSTR_TO_DWORD : BOOL //Return value TRUE = successful converted / FALSE if there are no valid hex signs or seperators
VAR_INPUT
	Hexstring 												: T_MaxString;
END_VAR
VAR_IN_OUT
{attribute 'displaymode':='hexadecimal'}
	Target													: DWORD;
END_VAR
VAR
	HexMarkerFound											: BOOL;
	i,j,Max_i,Max_j											: INT;
{attribute 'displaymode':='hexadecimal'}
	X														: BYTE;
{attribute 'displaymode':='hexadecimal'}
	TmpTarget												: DWORD;
END_VAR

Max_i 														:= LEN(Hexstring) - 1;
Max_j														:= SIZEOF(Target) * 2;
TmpTarget													:= 0;
HEXSTR_TO_DWORD												:= TRUE;
FOR i := 0 TO Max_i DO
	(* read the first character and subtract 48 to get value in decimal 0 = 48 *)
	(* calculate the value of the digit *)
	X														:= Hexstring[i];
	IF j >= Max_j
	THEN
		EXIT;
	ELSIF X > 47 AND x < 58 
	THEN //x = number 0-9
		TmpTarget 											:= SHL(TmpTarget,4) + X - 48;
		j													:= j + 1;
	ELSIF X > 64 AND X < 71 								
	THEN //x = letter A-F                   								
		TmpTarget 											:= SHL(TmpTarget,4) + X - 55;
		j													:= j + 1;
	ELSIF X > 96 AND X < 103								 
	THEN //x = letter a-f                     								
		TmpTarget 											:= SHL(TmpTarget,4) + X - 87;
		j													:= j + 1;
	ELSIF x = 16#58 OR x = 16#78 OR  x = 16#23
	THEN //found x, X or #, start over again because of 0xFA or 16#AB
		IF HexMarkerFound
		THEN
			HEXSTR_TO_DWORD									:= FALSE;	
			RETURN;		
		ELSE
			TmpTarget										:= 0;
			HexMarkerFound									:= TRUE;
			j												:= 0;	
		END_IF		
	ELSIF X = 16#2C OR X = 16#3A OR X = 16#2E OR X = 16#3B OR X = 16#20 OR X = 16#5F
	THEN //Ignore comma,colon,dot,space,underline
		; 
	ELSE
		HEXSTR_TO_DWORD										:= FALSE;	
		RETURN;
	END_IF
END_FOR
Target														:= TmpTarget;

END_FUNCTION

// ---- POUs/StringHelper/HEXSTR_TO_LWORD.TcPOU
{attribute 'no_check'}
//Converts a hex string into a 64 bit LWORD number
FUNCTION HEXSTR_TO_LWORD : BOOL //Return value TRUE = successful converted / FALSE if there are no valid hex signs or seperators
VAR_INPUT
	Hexstring 												: T_MaxString;
END_VAR
VAR_IN_OUT
{attribute 'displaymode':='hexadecimal'}
	Target													: LWORD;
END_VAR
VAR
	HexMarkerFound											: BOOL;
	i,j,Max_i,Max_j											: INT;
{attribute 'displaymode':='hexadecimal'}
	X														: BYTE;
{attribute 'displaymode':='hexadecimal'}
	TmpTarget												: LWORD;
END_VAR

Max_i 														:= LEN(Hexstring) - 1;
Max_j														:= SIZEOF(Target) * 2;
TmpTarget 													:= 0;
HEXSTR_TO_LWORD												:= TRUE;
FOR i := 0 TO Max_i DO
	(* read the first character and subtract 48 to get value in decimal 0 = 48 *)
	(* calculate the value of the digit *)
	X														:= Hexstring[i];
	IF j >= Max_j
	THEN
		EXIT;
	ELSIF X > 47 AND x < 58 
	THEN //x = number 0-9
		TmpTarget 											:= SHL(TmpTarget,4) + X - 48;
		j													:= j + 1;
	ELSIF X > 64 AND X < 71 								
	THEN //x = letter A-F                   								
		TmpTarget 											:= SHL(TmpTarget,4) + X - 55;
		j													:= j + 1;
	ELSIF X > 96 AND X < 103								 
	THEN //x = letter a-f                     								
		TmpTarget 											:= SHL(TmpTarget,4) + X - 87;
		j													:= j + 1;
	ELSIF x = 16#58 OR x = 16#78 OR  x = 16#23
	THEN //found x, X or #, start over again because of 0xFA or 16#AB
		IF HexMarkerFound
		THEN
			HEXSTR_TO_LWORD									:= FALSE;	
			RETURN;		
		ELSE
			TmpTarget										:= 0;
			HexMarkerFound									:= TRUE;
			j												:= 0;	
		END_IF		
	ELSIF X = 16#2C OR X = 16#3A OR X = 16#2E OR X = 16#3B OR X = 16#20 OR X = 16#5F
	THEN //Ignore comma,colon,dot,space,underline
		; 
	ELSE
		HEXSTR_TO_LWORD										:= FALSE;	
		RETURN;
	END_IF
END_FOR
Target														:= TmpTarget;

END_FUNCTION

// ---- POUs/StringHelper/INSERT_EXT.TcPOU
{attribute 'no_check' := ''}
FUNCTION INSERT_EXT : T_MaxString //The function INSERT_EXT inserts STR2 into STR1 at every ITERATION_POS position e.g. /r/n
VAR_INPUT
	STR1													:T_MaxString; //Base string - Hint! The base string will cut off if iteration of insertions exceeded the size of the string variable 
	STR2													:T_MaxString; //Insert string 
	ITERATION_POS											: INT; //Insert iteration position 
END_VAR
VAR
	Length1,length2,i,iEnd									: INT;														
END_VAR

INSERT_EXT													:= STR1;
Length1														:= LEN(STR1);
Length2														:= LEN(STR2);
IF TO_UINT(Length1 + Length2) > SIZEOF(STR1)
	OR ITERATION_POS = 0
THEN
	;
ELSE
	iEnd													:= MAX(1,ABS(Length1 / ITERATION_POS));
	FOR i := 1 TO iEnd
	DO 
		INSERT_EXT											:= INSERT(INSERT_EXT,STR2,(i*ITERATION_POS) + ((i-1)*Length2));
	END_FOR
END_IF

END_FUNCTION

// ---- POUs/StringHelper/LWORD_TO_BINSTR_EXT.TcPOU
{attribute 'no_check' := ''}
FUNCTION LWORD_TO_BINSTR_EXT : T_MaxString //This function converts a decimal number into a binary string (base 2), where the digits are separated according to the selected mode 
//e.g. 1111000011110000 -> 1111_0000_1111_0000 
VAR_INPUT
	In														: LWORD;//The decimal number requiring conversion.
	Precision												: INT; //Minimum number of displayed digits (digits), filled up with 0 from left if significant digits are less then that
	Mode													: INT; //1=Separate high and low word / 2=Separate bytes / 3=Separate nibbles /ELSE no separation | Separator = Param.DOWRD_TO_XXXSTR_EXT_SEPARATOR
END_VAR
VAR													
END_VAR

LWORD_TO_BINSTR_EXT 										:= LWORD_TO_BINSTR(in,precision);

CASE mode OF
1:// Separate by low word and high word
	LWORD_TO_BINSTR_EXT										:= INSERT_EXT(LWORD_TO_BINSTR_EXT,PARAM.XWORD_TO_XXXSTR_EXT_SEPARATOR,16);
	
2://Separate by bytes
	LWORD_TO_BINSTR_EXT										:= INSERT_EXT(LWORD_TO_BINSTR_EXT,PARAM.XWORD_TO_XXXSTR_EXT_SEPARATOR,8);
	
3://Separate by nibble
	LWORD_TO_BINSTR_EXT										:= INSERT_EXT(LWORD_TO_BINSTR_EXT,PARAM.XWORD_TO_XXXSTR_EXT_SEPARATOR,4);
END_CASE

END_FUNCTION

// ---- POUs/StringHelper/LWORD_TO_HEXSTR_EXT.TcPOU
{attribute 'no_check' := ''}
FUNCTION LWORD_TO_HEXSTR_EXT : T_MaxString //This function converts a decimal number into a hexadecimal string (base 16)., where the hex signs are separated according to the selected mode 
//e.g. F0F0F0F0 -> F0_F0_F0_F0 
VAR_INPUT
	In														: LWORD;
	Precision												: INT;//Minimum number of displayed signs, filled up with 0 from left if significant digits are less then that
	LoCase													: BOOL;
	Mode													: INT; //1=parted by word, 2=parted by byte, 3=parted by nibble
END_VAR
VAR
END_VAR

LWORD_TO_HEXSTR_EXT 										:= LWORD_TO_HEXSTR(in,precision,loCase);
CASE mode OF
1:// Separate by low word and high word
	LWORD_TO_HEXSTR_EXT										:= INSERT_EXT(LWORD_TO_HEXSTR_EXT,PARAM.XWORD_TO_XXXSTR_EXT_SEPARATOR,4);
	
2://Separate by bytes
	LWORD_TO_HEXSTR_EXT										:= INSERT_EXT(LWORD_TO_HEXSTR_EXT,PARAM.XWORD_TO_XXXSTR_EXT_SEPARATOR,2);
	
3://Separate by nibble
	LWORD_TO_HEXSTR_EXT										:= INSERT_EXT(LWORD_TO_HEXSTR_EXT,PARAM.XWORD_TO_XXXSTR_EXT_SEPARATOR,1);
END_CASE

END_FUNCTION

// ---- POUs/StringHelper/replaceInWString.TcPOU
{attribute 'no_check'}
//Replace a part of a string with another string 
FUNCTION replaceInWString : BOOL
VAR_INPUT
	SearchStr												:	WSTRING(10); //e.g. '/r/n_
	ReplaceStr												:	WSTRING(10); //e.g. '-'
END_VAR             										
VAR_IN_OUT         										
	Strline													: 	WSTRING(MAX_STRING_LENGTH);
END_VAR             										
VAR                 	
	StrLen, i,pos											:	INT;
END_VAR

IF strline = "" 
THEN 
	replaceInWString										:= TRUE;
ELSE
	StrLen													:= WLEN(strline);
	FOR i := 0 TO StrLen
	DO
		pos 												:= WFIND(strline,SearchStr);
		IF pos >= 1 
		THEN
			strline											:= WREPLACE(strline,ReplaceStr,WLEN(SearchStr),pos);
		ELSE
			replaceInWString								:= i > 0; 
			EXIT;						
		END_IF	
	END_FOR
END_IF

END_FUNCTION

// ---- POUs/TimeHelper/Conversions/FILETIME_TO_DATE.TcPOU
FUNCTION FILETIME_TO_DATE : DATE //Converts 64bit T_FILETIME to DATE (D#1970-01-01)
VAR_INPUT
	IN														: T_FILETIME;
END_VAR
VAR
END_VAR

FILETIME_TO_DATE											:= DT_TO_DATE(FILETIME_TO_DT(IN));

END_FUNCTION

// ---- POUs/TimeHelper/Conversions/LREAL_TO_TIME_SEC.TcPOU
{attribute 'no_check'}
//Convert time in lreal format <s.ms> into time format 
FUNCTION LREAL_TO_TIME_SEC : TIME
VAR_INPUT
	 IN														: LREAL;
END_VAR
VAR
END_VAR

LREAL_TO_TIME_SEC 											:= LREAL_TO_TIME(IN * 1000.0);

END_FUNCTION

// ---- POUs/TimeHelper/Conversions/SYSTEMTIME_TO_TOD.TcPOU
FUNCTION SYSTEMTIME_TO_TOD : TIME_OF_DAY //Converts Systemtime (Timestruct) to TIME_OF_DAY (TOD#15:36:30.123)
VAR_INPUT
	IN													: TIMESTRUCT;
END_VAR
VAR
END_VAR

SYSTEMTIME_TO_TOD											:= UDINT_TO_TOD(IN.wMilliseconds 
																+ IN.wSecond * 1000
																+ IN.wMinute * 60000
																+ IN.wHour * 3600000);

END_FUNCTION

// ---- POUs/TimeHelper/Conversions/SYSTEMTIME_TO_DATE.TcPOU
FUNCTION SYSTEMTIME_TO_DATE : DATE //Converts Systemtime (Timestruct) to DATE (D#2020-06-02)
VAR_INPUT
	IN													: TIMESTRUCT;
END_VAR
VAR
END_VAR

SYSTEMTIME_TO_DATE										:= DT_TO_DATE(SYSTEMTIME_TO_DT(IN));

END_FUNCTION

// ---- POUs/TimeHelper/getTonCountdown.TcPOU
{attribute 'no_check'}
//Provides the countdown value of an TON timer
FUNCTION getTonCountdown : TIME
VAR_IN_OUT
	Timer													:	TON;
END_VAR
VAR
END_VAR

IF Timer.IN
	AND NOT Timer.Q
THEN
	getTonCountdown 										:= Timer.PT - Timer.ET;
ELSE
	getTonCountdown 										:= T#0MS;
END_IF

END_FUNCTION

// ---- POUs/TimeHelper/OntimeExt.TcPOU
{attribute 'no_check'}
//Ontime function with external counter variables via references 
FUNCTION_BLOCK OntimeExt
VAR_INPUT
	IN														: 	BOOL := FALSE;		//Start ontime counting 
	ResetTrig												: 	BOOL := FALSE;		//Reset all counter
	rHour													:	REFERENCE TO UDINT;	//Ontime counter of total houres
	rMinute													:	REFERENCE TO UDINT;	//Ontime counter of minutes until one hour expired
	rSecond													:	REFERENCE TO UDINT; //Ontime counter of seconds until one minute expired
END_VAR
VAR_OUTPUT
	Error													:	BOOL;				//Invalid input references 
END_VAR
VAR
	txSys													: 	TIME;
	tx														: 	DWORD := 0;
	last													: 	DWORD := 0;
	ms														:	DWORD := 0;
	Init													:	BOOL := FALSE;
END_VAR

IF NOT __ISVALIDREF(rHour)
	OR NOT __ISVALIDREF(rMinute)
	OR NOT __ISVALIDREF(rSecond)
THEN
	Error													:= TRUE;
	RETURN;                 								
ELSE                        									
	Error 													:= FALSE;
END_IF                      	

(* read system time *)
txSys 														:= TIME();
tx 															:= TIME_TO_DWORD(txSys);
        													
(* make sure the first cycle works correctly *)
IF ResetTrig 
THEN
	reset();
ELSIF IN 
	AND Init 
THEN
	(* add the current milliseconds *)
	ms 														:= (tx - last) + ms;
	IF ms >= 1000 
	THEN
		rSecond 											:= rSecond + 1;
		IF rSecond >= 60
		THEN
			rSecond											:= 0;
			rMinute											:= rMinute + 1;
			IF rMinute >= 60
			THEN
				rMinute										:= 0;
				rHour										:= rHour + 1;
			END_IF
	  	END_IF
		ms 													:= ABS(ms - 1000);
	END_IF;
ELSE
	;
END_IF

Init 														:= TRUE;
last 														:= tx;

METHOD PUBLIC reset : BOOL //Return value = TRUE if execution finished
VAR_INPUT
END_VAR
	last 													:= tx;
	rHour 													:= rMinute := rSecond := 0;
	reset													:= TRUE;
END_METHOD

END_FUNCTION_BLOCK

// ---- POUs/TimeHelper/SensorTimeoutCheck.TcPOU
{attribute 'no_check'}
//This function-block checks wheter a sensor ("IN") is to long or to short occupied, based on the values of time and velocity which are related to the lenght
//Used to detect jamped pieces on a conveyor or flickering sensors
FUNCTION_BLOCK SensorTimeoutCheck
VAR_INPUT
	Enable													:	BOOL := TRUE;	//Enable 
	In														: 	BOOL := FALSE;	//Sensor signal 
	ResetTrig												:	BOOL := FALSE;	//Ack an error
	Offset_msec												: 	TIME := T#0MS; //ms
	Offset_mm												: 	LREAL := 300.0; //mm
	LenghtMin												:	LREAL := 100.0; //mm
 	LenghtMax												:	LREAL := 1000.0; //mm
	Velo													:	LREAL := 1000.0; //mm/s 
END_VAR             										
VAR_OUTPUT          										
	ErrorMin												:	BOOL	:= 0;	//Error - IN signal is flickering
	ErrorMax												: 	BOOL	:= 0;	//Error - IN signal is to long TRUE, a sign for jammed material
	TimeInFree												:	TIME	:= T#0MS;
	TimeInOccupied											:	TIME	:= T#0MS;                                                                                                       
END_VAR             	
VAR                 	
	TON_ToMin 												: 	TON;
	TON_ToMax 												: 	TON;
	MemSysTime												:	TIME;
	Mem														:	BYTE := 0;
	CntToMin												:	BYTE	:= 0;
END_VAR

(* monitors the toggle-signal of a sensor		 				       	 V2.2		*)
(************************************************************************************)

(* abort if not enable ***********************************************)
IF NOT Enable	
	OR ErrorMin
	OR ErrorMax
THEN
	Mem.1													:= TRUE;
	IF ResetTrig 
	THEN 
		reset();	
	END_IF
	RETURN;
END_IF
	
(* runtime meassuring *************************************)
TON_ToMin(
	IN 	:= TRUE, 
	PT 	:= LREAL_TO_TIME( ((LenghtMin + Offset_mm) / MAX(1.0, ABS(Velo)) ) * 1000.0) + Offset_msec,
	Q	=> );
	
IF IN AND NOT Mem.0 
THEN
	IF NOT TON_ToMin.Q
	THEN
		CntToMin											:= CntToMin + 1;
	ELSE                                                    	
		CntToMin											:= 0;
	END_IF                                                  	
	ErrorMin												:= CntToMin >= 3;
	TON_ToMin(IN := FALSE);
	TimeInOccupied := T#0MS;
ELSIF NOT In AND Mem.0 
THEN	
	IF NOT TON_ToMin.Q
	THEN
		CntToMin											:= CntToMin + 1;
	ELSE
		CntToMin											:= 0;
	END_IF
	ErrorMin												:= CntToMin >= 3;
	TON_ToMin(IN := FALSE);
	TimeInFree := T#0MS;
END_IF
Mem.0														:= In;

(* runtime error ********************************)
TON_ToMax(
	IN 	:= In AND NOT Mem.1, 
	PT 	:= LREAL_TO_TIME( ((LenghtMax + Offset_mm) / MAX(1.0, ABS(Velo)) ) * 1000.0) + Offset_msec,
	Q	=> ErrorMax);

(* runtime meassuring **************************************************)	
IF Mem.1 
THEN 
	MemSysTime 												:= TIME(); 
END_IF

IF IN 
THEN 
	TimeInOccupied 											:= TimeInOccupied + (TIME() - MemSysTime);
ELSE
	TimeInFree 												:= TimeInFree + (TIME() - MemSysTime);
END_IF
MemSysTime													:= TIME();

(* reset restart ************************************)
Mem.1														:= FALSE;
(********************************************************************************)

METHOD PUBLIC reset : BOOL
VAR_INPUT
END_VAR
ErrorMin := ErrorMAx 								:= FALSE; 
reset												:= TRUE;
END_METHOD

END_FUNCTION_BLOCK

// ---- POUs/TimeHelper/systemtimeInWin.TcPOU
{attribute 'no_check'}
// retuns True if Low <= In <= High Timestruct datatypes inputs
// 0 value will except part of this comparison
FUNCTION systemtimeInWin : Bool
VAR_IN_OUT
	In														: TIMESTRUCT;
	Low														: TIMESTRUCT;
	High													: TIMESTRUCT;
END_VAR
VAR
	LowOK													: BOOL;
	HighOK													: BOOL;
END_VAR

systemtimeInWin												:= FALSE;
LowOK														:= FALSE;
HighOK														:= FALSE;

IF In.wYear > Low.wYear THEN
	LowOK													:= TRUE;
ELSIF In.wYear = Low.wYear THEN
	IF In.wMonth > Low.wMonth THEN
			LowOK											:= TRUE;
	ELSIF In.wMonth = Low.wMonth THEN
		IF In.wDay > Low.wDay THEN
			LowOK											:= TRUE;
		ELSIF In.wDay = Low.wDay THEN
			IF In.wDayOfWeek > Low.wDayOfWeek THEN
				LowOK										:= TRUE;
			ELSIF In.wDayOfWeek = Low.wDayOfWeek THEN
				IF In.wHour > Low.wHour THEN
					LowOK									:= TRUE;
				ELSIF In.wHour = Low.wHour THEN
					IF In.wMinute > Low.wMinute THEN
						LowOK								:= TRUE;
					ELSIF In.wMinute = Low.wMinute THEN
						IF In.wSecond > Low.wSecond THEN
							LowOK							:= TRUE;
						ELSIF In.wSecond = Low.wSecond THEN
							IF In.wMilliseconds >= Low.wMilliseconds THEN
								LowOK						:= TRUE;
							END_IF	// ms
						END_IF	//s
					END_IF	//min 
				END_IF	// h
			END_IF	// dow
		END_IF	// d
	END_IF	// M
END_IF	// Y

IF In.wYear < High.wYear THEN
	HighOK													:= TRUE;
ELSIF In.wYear = High.wYear
	OR_ELSE High.wYear = 0
THEN
	IF In.wMonth < High.wMonth THEN
			HighOK											:= TRUE;
	ELSIF In.wMonth = High.wMonth
		 OR_ELSE High.wMonth = 0
	THEN
		IF In.wDay < High.wDay THEN
			HighOK											:= TRUE;
		ELSIF In.wDay = High.wDay 
			OR_ELSE High.wDay = 0
		THEN
			IF In.wDayOfWeek < High.wDayOfWeek THEN
				HighOK										:= TRUE;
			ELSIF In.wDayOfWeek = High.wDayOfWeek 
				OR_ELSE High.wDayOfWeek = 0
			THEN
				IF In.wHour < High.wHour THEN
					HighOK									:= TRUE;
				ELSIF In.wHour = High.wHour 
					OR_ELSE High.wHour = 0
				THEN
					IF In.wMinute < High.wMinute THEN
						HighOK								:= TRUE;
					ELSIF In.wMinute = High.wMinute 
						OR_ELSE High.wMinute = 0
					THEN
						IF In.wSecond < High.wSecond THEN
							HighOK							:= TRUE;
						ELSIF In.wSecond = High.wSecond 
							OR_ELSE High.wSecond = 0
						THEN
							IF In.wMilliseconds <= High.wMilliseconds 
								OR_ELSE High.wMilliseconds = 0
							THEN
								HighOK						:= TRUE;
							END_IF	// ms
						END_IF	//s
					END_IF	//min 
				END_IF	// h
			END_IF	// dow
		END_IF	// d
	END_IF	// M
END_IF	// Y

systemtimeInWin												:= LowOK AND HighOK;

END_FUNCTION

// ---- POUs/TimeHelper/VeloLinearMeasurement.TcPOU
{attribute 'no_check'}
//Accumulates the covered distance based on the velocity input and the time IN is TRUE - used to detect jamped pieces on a conveyor
FUNCTION_BLOCK VeloLinearMeasurement
VAR_INPUT
	Enable													:	BOOL;	//Enable function (e.g. Conveyor on)
	ResetTrig												:	BOOL;	//Reset Q
	IN														:	BOOL; 	//Sensor input
	Velo													:	LREAL;  //mm/ms | m/s with FACTOR=1, m/min with FACTOR=16.666666666666668
	Factor													:	LREAL := 1.0;	//Used to convert "VELO" into mm/ms (e.g. 16.666666666666668 to convert m/min into mm/ms
END_VAR             										
VAR_OUTPUT          										
	Q														:	LREAL;	//Accumulated value in mm
END_VAR             										
VAR                 										
	tx														:	DWORD;
	last 													: 	DWORD;
	ms														: 	DWORD;
	mmProms													:	LREAL;
END_VAR


(* Get mm pro ms *)
mmProms 													:= VELO * FACTOR; 

(* read system time *)
tx 															:= TIME_TO_DWORD(TIME());

(* Sequence *)
IF ResetTrig THEN
	reset();
ELSIF IN AND Enable THEN
	(* add the current milliseconds *)
	ms 														:= (tx - last) + ms;
	Q 														:= ms * mmProms;
ELSE
	;
END_IF

(* Save last Cylcetime *)
last 														:= tx;

(**********************************************************************)

METHOD PUBLIC reset : bool //Return value = TRUE if execution finished
VAR_INPUT
END_VAR
Q 															:= 0;
ms 															:= 0;
reset													:= TRUE;
END_METHOD

END_FUNCTION_BLOCK
